// TIA Portal project "teo2" (V15.1)

(* hardware
DEVICE "S7-400 station_1"  S7-400 station
   slot 0: "UR1_0"  UR1  6ES7 400-1TA01-0AA0
   slot 2: "PLC_1"  CPU 414-3 DP  6ES7 414-3XM05-0AB0  V5.3
      slot 1: "Interfaz DP_1"  X2
      slot 2: "Interfaz MPI/DP_1"  X1
*)

// ===== PLC "PLC_1"  CPU 414-3 DP =====

VAR_GLOBAL   // PLC tag table "Tabla de variables estándar"
   "S1" AT %I0.0 : Bool;   // Sensor de presencia plataforma A
   "S2" AT %I0.1 : Bool;   // Sensor de presencia plataforma B
   "S3" AT %I0.2 : Bool;   // Sensor de presencia plataforma C
   "Caja G" AT %I0.3 : Bool;   // Caja Grande
   "Caja P" AT %I0.4 : Bool;   // Caja Pequeña
   "P1" AT %I0.5 : Bool;   // Posicionador 1
   "P2" AT %I0.6 : Bool;   // Posicionador 2
   "P3" AT %I0.7 : Bool;   // Posicionador 3
   "INICIO" AT %I1.0 : Bool;   // Inicia el proceso
   "MARCA1" AT %M0.0 : Bool;
   "MARCA2" AT %M0.1 : Bool;
   "MARCA3" AT %M0.2 : Bool;
   "MARCA4" AT %M0.3 : Bool;
   "MARCA5" AT %M0.4 : Bool;
   "MARCA6" AT %M0.5 : Bool;
   "MARCA7" AT %M0.6 : Bool;
   "MARCA8" AT %M0.7 : Bool;
   "MARCA9" AT %M1.0 : Bool;
END_VAR

ORGANIZATION_BLOCK "Main"   // OB1, LAD
TITLE = "Main Program Sweep (Cycle)"
{ S7_Optimized_Access := 'FALSE' }
VERSION : 0.1
   VAR_TEMP
      OB1_EV_CLASS : Byte;   // Bits 0-3 = 1 (Coming event), Bits 4-7 = 1 (Event class 1)
      OB1_SCAN_1 : Byte;   // 1 (Cold restart scan 1 of OB 1), 3 (Scan 2-n of OB 1)
      OB1_PRIORITY : Byte;   // Priority of OB Execution
      OB1_OB_NUMBR : Byte;   // 1 (Organization block 1, OB1)
      OB1_RESERVED_1 : Byte;   // Reserved for system
      OB1_RESERVED_2 : Byte;   // Reserved for system
      OB1_PREV_CYCLE : Int;   // Cycle time of previous OB1 scan (milliseconds)
      OB1_MIN_CYCLE : Int;   // Minimum cycle time of OB1 (milliseconds)
      OB1_MAX_CYCLE : Int;   // Maximum cycle time of OB1 (milliseconds)
      OB1_DATE_TIME : Date_And_Time;   // Date and time OB1 started
   END_VAR
BEGIN

REGION Network 1: Inicio del proceso - Continuación del proceso
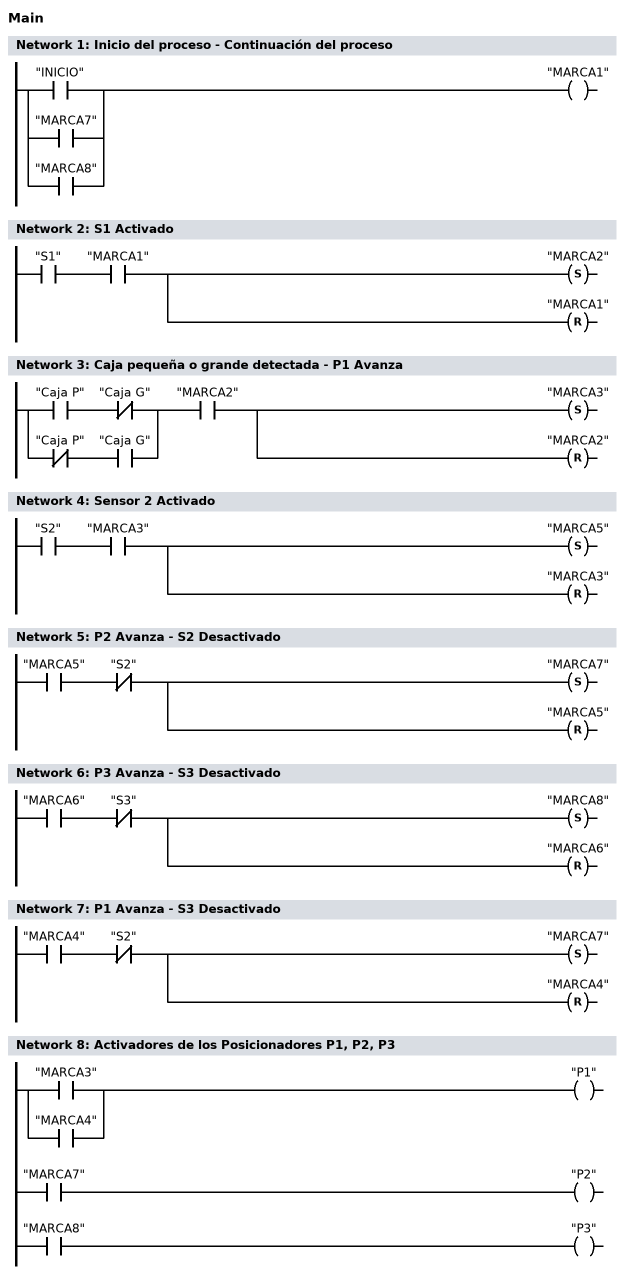
   RUNG wire#powerrail
      Contact( "INICIO" )
      wire#w1
      Coil( "MARCA1" )
   END_RUNG
   RUNG wire#powerrail
      Contact( "MARCA7" )
   END_RUNG wire#w1
   RUNG wire#powerrail
      Contact( "MARCA8" )
   END_RUNG wire#w1
   // the same network as SCL:
   "MARCA1" := "INICIO" OR "MARCA7" OR "MARCA8";
END_REGION

REGION Network 2: S1 Activado
   RUNG wire#powerrail
      Contact( "S1" )
      Contact( "MARCA1" )
      wire#w1
      S_Coil( "MARCA2" )
   END_RUNG
   RUNG wire#w1
      R_Coil( "MARCA1" )
   END_RUNG
   // the same network as SCL:
   IF "S1" AND "MARCA1" THEN
       "MARCA2" := TRUE;
       "MARCA1" := FALSE;
   END_IF;
END_REGION

REGION Network 3: Caja pequeña o grande detectada - P1 Avanza
   RUNG wire#powerrail
      Contact( "Caja P" )
      I_Contact( "Caja G" )
      wire#w1
      Contact( "MARCA2" )
      wire#w2
      S_Coil( "MARCA3" )
   END_RUNG
   RUNG wire#powerrail
      I_Contact( "Caja P" )
      Contact( "Caja G" )
   END_RUNG wire#w1
   RUNG wire#w2
      R_Coil( "MARCA2" )
   END_RUNG
   // the same network as SCL:
   IF (("Caja P" AND NOT "Caja G") OR (NOT "Caja P" AND "Caja G")) AND "MARCA2" THEN
       "MARCA3" := TRUE;
       "MARCA2" := FALSE;
   END_IF;
END_REGION

REGION Network 4: Sensor 2 Activado
   RUNG wire#powerrail
      Contact( "S2" )
      Contact( "MARCA3" )
      wire#w1
      S_Coil( "MARCA5" )
   END_RUNG
   RUNG wire#w1
      R_Coil( "MARCA3" )
   END_RUNG
   // the same network as SCL:
   IF "S2" AND "MARCA3" THEN
       "MARCA5" := TRUE;
       "MARCA3" := FALSE;
   END_IF;
END_REGION

REGION Network 5: P2 Avanza - S2 Desactivado
   RUNG wire#powerrail
      Contact( "MARCA5" )
      I_Contact( "S2" )
      wire#w1
      S_Coil( "MARCA7" )
   END_RUNG
   RUNG wire#w1
      R_Coil( "MARCA5" )
   END_RUNG
   // the same network as SCL:
   IF "MARCA5" AND NOT "S2" THEN
       "MARCA7" := TRUE;
       "MARCA5" := FALSE;
   END_IF;
END_REGION

REGION Network 6: P3 Avanza - S3 Desactivado
   RUNG wire#powerrail
      Contact( "MARCA6" )
      I_Contact( "S3" )
      wire#w1
      S_Coil( "MARCA8" )
   END_RUNG
   RUNG wire#w1
      R_Coil( "MARCA6" )
   END_RUNG
   // the same network as SCL:
   IF "MARCA6" AND NOT "S3" THEN
       "MARCA8" := TRUE;
       "MARCA6" := FALSE;
   END_IF;
END_REGION

REGION Network 7: P1 Avanza - S3 Desactivado
   RUNG wire#powerrail
      Contact( "MARCA4" )
      I_Contact( "S2" )
      wire#w1
      S_Coil( "MARCA7" )
   END_RUNG
   RUNG wire#w1
      R_Coil( "MARCA4" )
   END_RUNG
   // the same network as SCL:
   IF "MARCA4" AND NOT "S2" THEN
       "MARCA7" := TRUE;
       "MARCA4" := FALSE;
   END_IF;
END_REGION

REGION Network 8: Activadores de los Posicionadores P1, P2, P3
   RUNG wire#powerrail
      Contact( "MARCA3" )
      wire#w1
      Coil( "P1" )
   END_RUNG
   RUNG wire#powerrail
      Contact( "MARCA4" )
   END_RUNG wire#w1
   RUNG wire#powerrail
      Contact( "MARCA7" )
      Coil( "P2" )
   END_RUNG
   RUNG wire#powerrail
      Contact( "MARCA8" )
      Coil( "P3" )
   END_RUNG
   // the same network as SCL:
   "P1" := "MARCA3" OR "MARCA4";
   "P2" := "MARCA7";
   "P3" := "MARCA8";
END_REGION
END_ORGANIZATION_BLOCK